TYPE STATE:
    STRUCT
        curTime: LREAL;
        dvar_M_p: DINT;
    END_STRUCT;
END_TYPE
